Yaskawa INFORM job: CLEAN-R1_KM_NEW_SCIANA.JBI

/JOB
//NAME CLEAN-R1_KM_NEW_SCIANA
///FOLDERNAME CLEAN
//POS
///NPOS 26,26,0,2,0,0
///TOOL 0
///POSTYPE PULSE
///PULSE
C00000=2508,0,0,0,0,4169
C00001=41115,93452,-30342,-19926,115521,85678
C00002=28599,109925,-13759,-12658,112881,84157
C00003=28878,100235,-19265,-13345,108164,84179
C00004=28966,99224,-20084,-13542,107459,84155
C00005=29027,99166,-20392,-13590,107618,84144
C00006=28599,108424,-14443,-12622,112541,84195
C00007=23674,85929,9201,-23424,39910,87231
C00008=22849,91751,19297,-24107,36761,87842
C00009=22769,92475,20456,-24200,36429,87915
C00010=27413,53480,-29931,-24215,47505,86509
C00011=23674,85929,9201,-23424,39910,87231
C00012=28599,108424,-14443,-12622,112541,84195
C00013=34011,109773,-12073,-16636,107751,84808
C00014=32816,112629,-5671,-14598,109695,85231
C00015=32618,110353,-5730,-14378,108579,85337
C00016=32545,109523,-5728,-14298,108158,85375
C00017=32618,110353,-5730,-14378,108579,85337
C00018=32816,112629,-5671,-14598,109695,85231
C00019=34011,109773,-12073,-16636,107751,84808
C00020=38810,111241,-7992,-19438,105697,85727
C00021=36913,114349,813,-16982,106196,86149
C00022=37169,116704,797,-17245,107389,86018
C00023=39968,92120,-23778,-21749,94252,85800
C00024=46315,71110,-54300,-23622,119041,85704
C00025=32571,-80067,-84751,-11816,58952,90735
BC00000=0,0,0
BC00001=204899,578,1075157
BC00002=204899,578,1075157
BC00003=204899,578,1075157
BC00004=204899,578,1075157
BC00005=204899,578,1075157
BC00006=204899,578,1075157
BC00007=125260,578,1075157
BC00008=125260,578,1075157
BC00009=125260,578,1075157
BC00010=125260,578,1075155
BC00011=125260,578,1075157
BC00012=204899,578,1075157
BC00013=204899,578,1075157
BC00014=204899,578,1075157
BC00015=204899,578,1075157
BC00016=204899,578,1075157
BC00017=204899,578,1075157
BC00018=204899,578,1075157
BC00019=204899,578,1075157
BC00020=204899,578,1075157
BC00021=204894,578,1075156
BC00022=204894,578,1075156
BC00023=204894,578,1075156
BC00024=204899,578,1075157
BC00025=204899,578,820586
///POSTYPE BASE
///RECTAN
///RCONF 0,0,0,0,1,0,0,0,0,0,0,0,0,0,0,0,0,0,0,0,0,0,0,0
P00122=3137.544,3958.137,1922.667,15.5192,-68.1197,-17.3024
P00123=0.398,-92.365,-0.154,0.0099,0.0024,-0.0079
//INST
///DATE 2024/07/16 19:47
///ATTR SC,RW
///GROUP1 RB1,BS1
///LVARS 0,5,5,1,0,3,3,0
NOP
INC B060
SET I010 B060
MUL I010 100
DIV I010 56
SFTOF
SFTOF3D
SET B050 0
JUMP *START
*BEGIN
SET B050 2
*START
'********************************
'Please check position before
'running in play-mode
'********************************
'#Output - Cleaning Motor
SET LI000 14
'#Output - Cleaning Oil
SET LI001 15
'#Output - Wirecut
SET LI002 16
'#Output - Wirefeeder Forward
SET LI003 4095
'#Output - Torch Blow out
SET LI004 4091
'********************************
REFP 1 C00000 BC00000
GETS LPX001 $PX011
CNVRT LPX001 LPX001 RF
GETS LPX002 $PX001
CNVRT LPX002 LPX002 RF
SUB LBP002 LBP001
'Comment out axis to shift
SETE LBP002 (1) 0
COMM SETE LBP002 (2) 0
SETE LBP002 (3) 0
SFTON LBP002
'********************************
'SAFE POS
PAUSE IF IN#(1563)=OFF
MOVJ C00001 BC00001 VJ=100.00
'WIRECUT
MOVJ C00002 BC00002 VJ=100.00
DOUT OT#(LI003) OFF
DOUT OT#(LI002) OFF
'WIREFEED OUTPUT
MOVL C00003 BC00003 V=133.3
COMM PULSE OT#(LI003) T=0.80
DOUT OT#(LI003) ON
TIMER T=0.90
DOUT OT#(LI003) OFF
TIMER T=0.50
MOVL C00004 BC00004 V=20.0
TIMER T=1.00
DOUT OT#(LI002) ON
TIMER T=1.00
DOUT OT#(LI002) OFF
MOVL C00005 BC00005 V=20.0
MOVL C00006 BC00006 V=166.7
'CHECK
MOVL C00007 BC00007 V=166.7 PL=1
MOVL C00008 BC00008 V=166.7 PL=0
MOVL C00009 BC00009 V=8.3 SRCH RIN#(1)=ON DIS=20.0
GETS PX123 $PX001
SUB P123 P122
GETE LD000 P123 (1)
GETE LD002 P123 (3)
MUL LD000 LD000
MUL LD002 LD002
ADD LD000 LD002
SET LR000 LD000
DIV LR000  1.000000E+06
SQRT LR000 LR000
IFTHENEXP LR000> 1.000000E+00
	 MOVL C00010 BC00010 V=83.3
	 JUMP *BEGIN IF B050<2
	 IFTHENEXP B050=2
		 SETUALM 8201 "PROBLEM DL DRUTU" 0
		 JUMP *BEGIN
	 ENDIF
ENDIF
DOUT OT#(LI002) OFF
'CLEANING MOTOR
MOVL C00011 BC00011 V=166.7
MOVL C00012 BC00012 V=166.7 PL=1
MOVJ C00013 BC00013 VJ=100.00
MOVL C00014 BC00014 V=166.7
'CLEANING AIR
DOUT OT#(LI004) ON
MOVL C00015 BC00015 V=20.0
TIMER T=0.20
DOUT OT#(LI000) ON
TIMER T=0.50
MOVL C00016 BC00016 V=20.0
TIMER T=0.50
MOVL C00017 BC00017 V=20.0
TIMER T=0.20
DOUT OT#(LI000) OFF
TIMER T=0.50
DOUT OT#(LI004) OFF
MOVL C00018 BC00018 V=83.3
MOVL C00019 BC00019 V=166.7
'CLEANING OIL
MOVJ C00020 BC00020 VJ=100.00
JUMP *111
MOVL C00021 BC00021 V=166.7
PULSE OT#(LI001) T=0.20
TIMER T=1.00
MOVL C00022 BC00022 V=250.0
'CLEANING AIR
PULSE OT#(LI004) T=1.00
TIMER T=1.00
MOVJ C00023 BC00023 VJ=50.00
'SAFE POS
*111
MOVJ C00024 BC00024 VJ=100.00
MOVJ C00025 BC00025 VJ=100.00
SFTOF
SFTOF3D
SFTOF
'********************************
'*         CLEANING JOB         *
'*      __ __ _____ _____       *
'*     |  |  |   | | __  |      *
'*     |_   _| | | |    -|      *
'*       |_| |_|___|__|__|      *
'*        YRC Multi Base        *
'*       rev 4. 2021-10-12      *
'********************************
END
